FUNCTION WithinTolerance : BOOL
VAR_INPUT
	v1 : LREAL;
	v2 : LREAL;
	tolerance : LREAL;
END_VAR

WithinTolerance := ABS(v1-v2) < tolerance;

END_FUNCTION

(* stored: Version 1.1.0.1, ProductVersion 3.1.4024.11
   POU WithinTolerance: Id {5a9723bf-6f01-425f-91fc-113cb1f94a16}, SpecialFunc None *)
